// TIA Portal V21 export
DATA_BLOCK "RETAIN"   // DB81
{ S7_Optimized_Access := 'FALSE' }
   VAR RETAIN
      "CHAMBER PRESS SCL MAX" : Real := 5.0;
      "CHAMBER PRESS SCL MIN" : Real := -1.0;
      "JACKET PRESS SCL MAX" : Real := 5.0;
      "JACKET PRESS SCL MIN" : Real := -1.0;
      "CHAMBER VCC SCL MAX" : Real := 5.0;
      "CHAMBER VCC SCL MIN" : Real := -1.0;
      "SET PWD TEMP" : Real := 0.0;
      "SET CHAMBER PRESS HIGH" : Real := 1.25;
      "SET STERILE TEMP1" : Real := 105.0;
      "SET DRY VCC" : Real := -0.5;
      "SET STERILE EXH PRESS" : Real := 0.05;
      "SET ATM PRESS" : Real := -0.05;
      "SET EXIT TEMP" : Real := 101.0;
      "SET CHAMBER PRESS LOW" : Real := 1.18;
      "SET WFI TEMP" : Real := 0.0;
      "SET CONTROL BAND" : Real := 0.2;
      "SET STERILE TEMP2" : Real := 110.0;
      "SET STERILE TEMP3" : Real := 115.0;
      "SET STERILE TEMP4" : Real := 121.4;
      "SET LEAK VCC" : Real := -0.7;
      "SET VCC PRESS" : Real := -0.05;
      "SET STD1 TEMP1" : Real := 100.0;
      "SET STD1 TEMP2" : Real := 110.0;
      "SET STD1 TEMP3" : Real := 119.0;
      "SET STD1 PRESS" : Real := 0.05;
      "SET BOW VCC" : Real := -0.6;
      "SET BOW HEATUP" : Real := 121.4;
      "SET BOW EXH PRESS" : Real := 0.05;
      "SET BOW ATS PRESS" : Real := 0.0;
      "SET BOW END PRESS" : Real := -0.05;
      "SET BOW UP PRESS" : Real := 0.5;
      "SET HPHV VCC" : Real := -0.6;
      "SET HPHV HEATUP" : Real := 121.4;
      "SET HPHV EXH PRESS" : Real := 0.5;
      "SET HPHV ATS PRESS" : Real := -0.5;
      "SET HPHV END PRESS" : Real := -0.05;
      "SET HPHV UP PRESS" : Real := 0.5;
      "SET HZ" : Real := 25.0;
      "DOOR1 VCC SCL MIN" : Real := -1.0;
      "DOOR1 VCC SCL MAX" : Real := 5.0;
      "DOOR2 VCC SCL MIN" : Real := -1.0;
      "DOOR2 VCC SCL MAX" : Real := 5.0;
      "DOOR1 PRESS SCL MIN" : Real := -1.0;
      "DOOR1 PRESS SCL MAX" : Real := 5.0;
      "DOOR2 PRESS SCL MIN" : Real := -1.0;
      "DOOR2 PRESS SCL MAX" : Real := 5.0;
      "SET JACKET PRESS HIGH" : Real := 1.25;
      "SET DOOR1 PRESS HIGH" : Real := 2.55;
      "SET DOOR2 PRESS HIGH" : Real := 2.55;
      "SET DOOR1 VCC" : Real := -0.7;
      "SET DOOR2 VCC" : Real := -0.7;
      "SET JACKET LOW PRESS" : Real := 1.1;
      "SET DOOR1 PRESS LOW" : Real := 2.35;
      "SET DOOR2 PRESS LOW" : Real := 2.35;
      "SET PWD INLET TIME" : Int := 7;
      "SET DTG DSG TIME" : Int := 60;
      "SET PWD CRC TIME" : Int := 10;
      "SET PWD DRAIN" : Int := 7;
      "SET PRINT INTERVAL" : Int := 60;
      "SET WFI INLET TIME" : Int := 7;
      "SET WFI DSG TIME" : Int := 60;
      "SET WFI CRC TIME" : Int := 10;
      "SET WFI DRAIN TIME" : Int := 10;
      "SET WFI COUNTS" : Int := 0;
      "SET STERILE TIME1" : Int := 5;
      "SET STERILE TIME2" : Int := 5;
      "SET STERILE TIME3" : Int := 5;
      "SET STERILE TIME4" : Int := 30;
      "SET VENT TIME" : Int := 0;
      "SET VCC HOLD TIME" : Int := 10;
      "SET STD1 HOLD1" : Int := 5;
      "SET STD1 HOLD2" : Int := 3;
      "SET STD1 HOLD3" : Int := 2;
      "SET BOW  VCC HOLD TIME" : Int := 0;
      "SET NO OF BOW" : Int := 4;
      "SET BOW HEAT HOLD TIME" : Int := 10;
      "SET BOW ATS HOLD" : Int := 0;
      "SET DRY TIME" : Int := 20;
      "SET HPHV VCC HOLD" : Int := 0;
      "SET NO OF HPHV" : Int := 3;
      "SET HPHV HEAT HOLD" : Int := 10;
      "SET HPHV ATS HOLD" : Int := 5;
      "SET NO OF PWD" : Int := 2;
      "SET OFF EXHAUST" : Int := 40;
      "SET ON EXHAUST" : Int := 2;
      "SET STD1 VCC" : Real := 0.0;
      "SET STD1 UP PRESS" : Real := 0.0;
      "SET STD1 VCC HOLD" : Int := 0;
      "SET NO OF STD1 PULSE" : Int := 0;
      "SET STD2 TEMP1" : Real := 100.0;
      "SET STD2 TEMP2" : Real := 110.0;
      "SET STD2 TEMP3" : Real := 119.0;
      "SET STD2 PRESS" : Real := 0.05;
      "SET STD2 HOLD1" : Int := 5;
      "SET STD2 HOLD2" : Int := 3;
      "SET STD2 HOLD3" : Int := 2;
      "SET STD2 VCC" : Real := 0.0;
      "SET STD2 UP PRESS" : Real := 0.0;
      "SET STD2 VCC HOLD" : Int := 0;
      "SET NO OF STD2 PULSE" : Int := 0;
      "SET ACCEPTANCE LEAK" : Real := 0.013;
      "JACKET VCC SCL MIN" : Real := -1.0;
      "JACKET VCC SCL MAX" : Real := 5.0;
      "SET DELAY BEFORE HOLD" : Int := 3;
      "SET OVERSHOOT" : Real := 124.0;
      "SET ABORT TEMP" : Real := 120.5;
      DUMMY2 : Real := 0.0;
      DUMMY3 : Real := 0.0;
      DUMMY4 : Real := 0.0;
      DUMMY5 : Real := 0.0;
      DUMMY6 : Real := 0.0;
      "SET ABORT DELAY" : Int := 0;
      "SET WFI NO OF CYCLE" : Int := 0;
      "INT ATG3" : Int := 0;
      "INT ATG4" : Int := 0;
      "INT ATG5" : Int := 0;
      "INT ATG6" : Int := 0;
      "INT ATG7" : Int := 0;
      "INT ATG8" : Int := 0;
      "INT ATG9" : Int := 0;
      STD3 { S7_SetPoint := 'True'} : "STD";
      STD4 { S7_SetPoint := 'True'} : "STD";
      STD5 { S7_SetPoint := 'True'} : "STD";
      STD6 { S7_SetPoint := 'True'} : "STD";
      STD7 { S7_SetPoint := 'True'} : "STD";
      STD8 { S7_SetPoint := 'True'} : "STD";
      STD9 { S7_SetPoint := 'True'} : "STD";
      "SET BOILER ON TEMP" : Real := 133.0;
      "SET BOILER OFF TEMP" : Real := 135.0;
      "SET JACKET ON TIME" : Int := 10;
      "SET JACKET OFF TIME" : Int := 10;
      "SET BOILER WATER OFF DELAY" : Int := 25;
      "SET PRESSURE VERY HIGH" : Real := 1.3;
      "SET VACUUM BREAK FAIL TIME" : Int := 10;
      "SET JACKET PRESSURE HH" : Real := 1.4;
      "SET DOOR1 ALM PRESSURE" : Real := 0.3;
      "SET DOOR2 ALM PRESSURE" : Real := 0.3;
   END_VAR
BEGIN
   STD3."SET TEMP1" := 0.0;
   STD3."SET TEMP2" := 0.0;
   STD3."SET TEMP3" := 0.0;
   STD3."SET PRESS" := 0.0;
   STD3."SET HOLD1" := 0;
   STD3."SET HOLD2" := 0;
   STD3."SET HOLD3" := 0;
   STD3."SET VCC" := 0.0;
   STD3."SET UP PRESS" := 0.0;
   STD3."SET VCC HOLD" := 0;
   STD3."SET NO OF PULSE" := 0;
   STD4."SET TEMP1" := 0.0;
   STD4."SET TEMP2" := 0.0;
   STD4."SET TEMP3" := 0.0;
   STD4."SET PRESS" := 0.0;
   STD4."SET HOLD1" := 0;
   STD4."SET HOLD2" := 0;
   STD4."SET HOLD3" := 0;
   STD4."SET VCC" := 0.0;
   STD4."SET UP PRESS" := 0.0;
   STD4."SET VCC HOLD" := 0;
   STD4."SET NO OF PULSE" := 0;
   STD5."SET TEMP1" := 0.0;
   STD5."SET TEMP2" := 0.0;
   STD5."SET TEMP3" := 0.0;
   STD5."SET PRESS" := 0.0;
   STD5."SET HOLD1" := 0;
   STD5."SET HOLD2" := 0;
   STD5."SET HOLD3" := 0;
   STD5."SET VCC" := 0.0;
   STD5."SET UP PRESS" := 0.0;
   STD5."SET VCC HOLD" := 0;
   STD5."SET NO OF PULSE" := 0;
   STD6."SET TEMP1" := 0.0;
   STD6."SET TEMP2" := 0.0;
   STD6."SET TEMP3" := 0.0;
   STD6."SET PRESS" := 0.0;
   STD6."SET HOLD1" := 0;
   STD6."SET HOLD2" := 0;
   STD6."SET HOLD3" := 0;
   STD6."SET VCC" := 0.0;
   STD6."SET UP PRESS" := 0.0;
   STD6."SET VCC HOLD" := 0;
   STD6."SET NO OF PULSE" := 0;
   STD7."SET TEMP1" := 0.0;
   STD7."SET TEMP2" := 0.0;
   STD7."SET TEMP3" := 0.0;
   STD7."SET PRESS" := 0.0;
   STD7."SET HOLD1" := 0;
   STD7."SET HOLD2" := 0;
   STD7."SET HOLD3" := 0;
   STD7."SET VCC" := 0.0;
   STD7."SET UP PRESS" := 0.0;
   STD7."SET VCC HOLD" := 0;
   STD7."SET NO OF PULSE" := 0;
   STD8."SET TEMP1" := 0.0;
   STD8."SET TEMP2" := 0.0;
   STD8."SET TEMP3" := 0.0;
   STD8."SET PRESS" := 0.0;
   STD8."SET HOLD1" := 0;
   STD8."SET HOLD2" := 0;
   STD8."SET HOLD3" := 0;
   STD8."SET VCC" := 0.0;
   STD8."SET UP PRESS" := 0.0;
   STD8."SET VCC HOLD" := 0;
   STD8."SET NO OF PULSE" := 0;
   STD9."SET TEMP1" := 0.0;
   STD9."SET TEMP2" := 0.0;
   STD9."SET TEMP3" := 0.0;
   STD9."SET PRESS" := 0.0;
   STD9."SET HOLD1" := 0;
   STD9."SET HOLD2" := 0;
   STD9."SET HOLD3" := 0;
   STD9."SET VCC" := 0.0;
   STD9."SET UP PRESS" := 0.0;
   STD9."SET VCC HOLD" := 0;
   STD9."SET NO OF PULSE" := 0;
END_DATA_BLOCK
